{attribute 'linkalways'} 
{attribute 'no_explicit_call' := 'This FB is a CLASS and must be accessed using methods or properties'}
{attribute 'enable_dynamic_creation'}
FUNCTION_BLOCK Node_F_VN_GetAt_TcVnVector4_DINT EXTENDS VisionNode
VAR
    ipContainer : _ITcVnContainer;
    aElement : _TcVnVector4_DINT;
    nIndex : _ULINT(0);
    hrPrev : _HRESULT(S_OK);
    hresult : _HRESULT(S_OK);
END_VAR

METHOD PUBLIC  Clone : I_Node
VAR
	pNode : POINTER TO Node_F_VN_GetAt_TcVnVector4_DINT;
END_VAR
pNode := __NEW(Node_F_VN_GetAt_TcVnVector4_DINT);
Clone := pNode^;
END_METHOD

METHOD FB_init : BOOL
VAR_INPUT
	bInitRetains : BOOL; // if TRUE, the retain variables are initialized (warm start / cold start)
	bInCopyCode : BOOL;  // if TRUE, the instance afterwards gets moved into the copy code (online change)
END_VAR
AddInput('ipContainer', ipContainer);
AddParameter('nIndex', nIndex);
AddInput('hrPrev', hrPrev);
AddOutput('aElement', aElement);
AddOutput('hresult',hresult);
END_METHOD

METHOD PROTECTED OnExecute
hresult.Value := F_VN_GetAt_TcVnVector4_DINT(
    ipContainer := ipContainer.Value,
    aElement := aElement.Value,
    nIndex := nIndex.Value,
    hrPrev:= hrPrev.Value);
END_METHOD

METHOD PUBLIC PreExecutionCheck
VAR_INPUT
	Check : I_PreExecutionChecks;
END_VAR
Check.IsTrue(ipContainer.IsValid, 'ipContainer must be a valid container');
Check.IsTrue(ipContainer.IsType(TC_GLOBAL_CONST_LIST.ContainerType_Vector_TcVnVector4_DINT), 'ipContainer contains incorrect type');
END_METHOD

END_FUNCTION_BLOCK

(* stored: Version 1.1.0.1, ProductVersion 3.1.4026.13
   POU Node_F_VN_GetAt_TcVnVector4_DINT: Id {4e110cff-d387-47a3-9e1e-72de85fd25c0}, SpecialFunc None
   Folder Constructor: Id {56ac77be-084f-4143-a6c9-f4458c393ca9}
   Method Clone: Id {1a21154d-7c0c-45be-bc14-b906800dd26e}
   Method FB_init: Id {268f7652-531e-482f-95d6-aea326f5c96d}
   Method OnExecute: Id {5b5c36ed-2e27-4cf0-962b-b07aaf562051}
   Method PreExecutionCheck: Id {a064f6b7-f58b-4fe9-9dba-9c0f6ea85ab9} *)
